FUNCTION_BLOCK ATM_IN_US_TO_ADI (* Convert TIME (via ATM adapter) in US to DINT (via ADI adapter) *)
  (* Standard: 61499-2; Description: Copyright (c) 2026 HR Agrartechnik GmbH This program and the accompanying materials are made available under the terms of the Eclipse Public License 2.0 which is available at https://www.eclipse.org/legal/epl-2.0/ SPDX-License-Identifier: EPL-2.0 *)
  (* Version 1.0, 2026-08-13, Franz Höpfinger, HR Agrartechnik GmbH, initial API and implementation *)
  PACKAGE adapter::conversion::unidirectional;
  IMPORT iec61131::conversion::F_TIME_IN_US_TO_DINT;
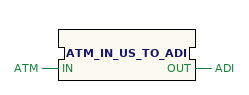
  SOCKETS
    IN : adapter::types::unidirectional::ATM; (* Time value to convert *)
  END_SOCKETS
  PLUGS
    OUT : adapter::types::unidirectional::ADI; (* TIME value of IN expressed in US as DINT *)
  END_PLUGS
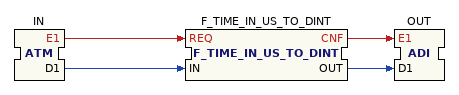
  FBS
    F_TIME_IN_US_TO_DINT : iec61131::conversion::F_TIME_IN_US_TO_DINT;
  END_FBS
  EVENT_CONNECTIONS
    IN.E1 TO F_TIME_IN_US_TO_DINT.REQ;
    F_TIME_IN_US_TO_DINT.CNF TO OUT.E1;
  END_CONNECTIONS
  DATA_CONNECTIONS
    IN.D1 TO F_TIME_IN_US_TO_DINT.IN;
    F_TIME_IN_US_TO_DINT.OUT TO OUT.D1;
  END_CONNECTIONS
END_FUNCTION_BLOCK
